// TIA Portal V16 export
// export: Created 2024-05-10T06:46:43.1229675Z, ExportSetting WithDefaults, DisplayName Totally Integrated Automation Portal, DisplayVersion V16, DisplayName TIA Portal Version Control Interface, DisplayVersion V16, DisplayName TIA Portal Openness, DisplayVersion V16, DisplayName STEP 7 Professional, DisplayVersion V16, DisplayName STEP 7 Safety, DisplayVersion V16, DisplayName WinCC Professional, DisplayVersion V16
FUNCTION_BLOCK "F121_SinaParaWrite(SV660F)"   // FB121, LAD
{ S7_Optimized_Access := 'TRUE' }
VERSION : 0.1
// stored: AutoNumber false, IsIECCheckEnabled false, IsRetainMemResEnabled false, MemoryReserve 100, SetENOAutomatically false, UDAEnableTagReadback false
   VAR_INPUT
      ID_回原高速 : DInt;
      ID_回原低速 : DInt;
      ID_点动速度 : DInt;
      ID_最高速度 : DInt;
      IM_故障复位 : Bool;
      ID_111报文标识符 { ExternalAccessible := 'False'; ExternalVisible := 'False'; ExternalWritable := 'False'} : HW_IO;
   END_VAR
   VAR_OUTPUT
      OM_准备好 : Bool;
      OM_进行中 : Bool;
      OM_正常完了 : Bool;
      OR_数据Real : Real;
      OD_数据Dint : DInt;
      OW_数据格式 : Int;
      OW_故障码 : Int;
      OM_故障 : Bool;
      OW_SFB调用错误 : Word;
   END_VAR
   VAR
      MT_Time { ExternalAccessible := 'False'; ExternalVisible := 'False'; ExternalWritable := 'False'} : IEC_TIMER;
   END_VAR
   VAR_TEMP
      MD_回原高速 : Array[1..2] of DInt;
      MD_回原低速 : Array[1..2] of DInt;
      MD_点动正速度 : Array[1..2] of DInt;
      MD_点动负速度 : Array[1..2] of DInt;
      MD_最高速度 : Array[1..2] of DInt;
      M_回原高速变更 : Bool;
      M_回原低速变更 : Bool;
      M_点动正速度变更 : Bool;
      M_点动负速度变更 : Bool;
      M_最高速度变更 : Bool;
      M_回原高速写入 : Bool;
      M_回原低速写入 : Bool;
      M_点动正速度写入 : Bool;
      M_点动负速度写入 : Bool;
      M_最高速度写入 : Bool;
      M_开始 : Bool;
      MW_Parameter : Int;
      MW_Index : Int;
      MD_Value : DInt;
      M_Pulse : Array[1..2] of Bool;
   END_VAR
   VAR_TEMP   // added for the SCL form of the ladder/FBD networks
      _w1 : Bool;
      _w2 : Bool;
      _w3 : Bool;
      _w4 : Bool;
      _w5 : Bool;
      _w6 : Bool;
   END_VAR
BEGIN

REGION Network 1: 回原高速
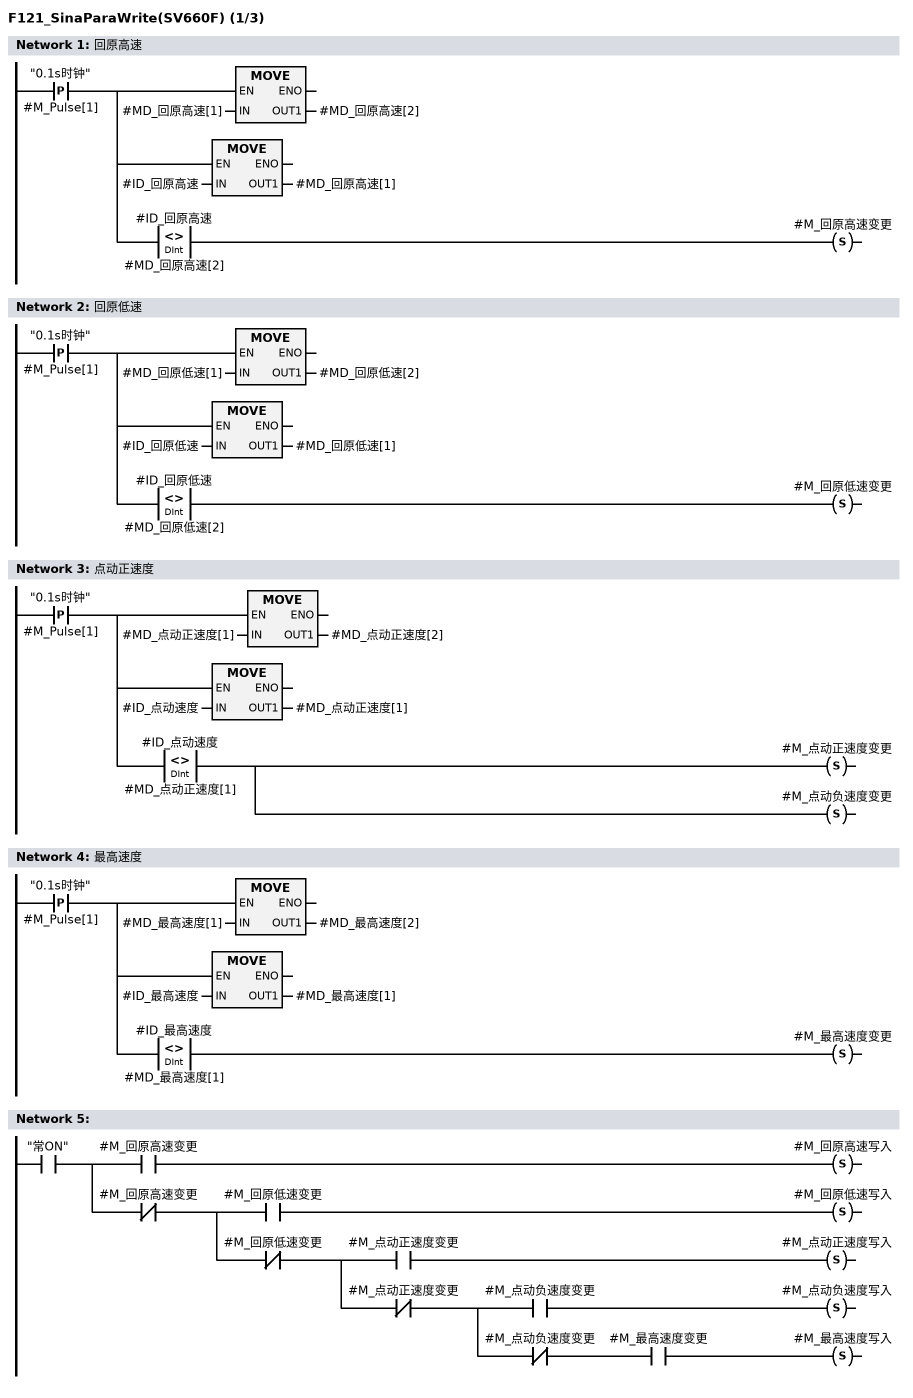
   RUNG wire#powerrail
      P_Contact(operand := "0.1s时钟", bit := #M_Pulse[1])
      wire#w1
      Move(in := #MD_回原高速[1], out1 => #MD_回原高速[2])
   END_RUNG
   RUNG wire#w1
      Move(in := #ID_回原高速, out1 => #MD_回原高速[1])
   END_RUNG
   RUNG wire#w1
      { S7_Templates := "SrcType := DInt" } NE_Contact(in1 := #ID_回原高速, in2 := #MD_回原高速[2])
      S_Coil( #M_回原高速变更 )
   END_RUNG
   // the same network as SCL:
   #_w1 := "0.1s时钟" AND NOT #M_Pulse[1];   // rising edge of "0.1s时钟"
   #M_Pulse[1] := "0.1s时钟";
   IF #_w1 THEN
       #MD_回原高速[2] := #MD_回原高速[1];
       #MD_回原高速[1] := #ID_回原高速;
   END_IF;
   IF #_w1 AND (#ID_回原高速 <> #MD_回原高速[2]) THEN #M_回原高速变更 := TRUE; END_IF;
END_REGION

REGION Network 2: 回原低速
   RUNG wire#powerrail
      P_Contact(operand := "0.1s时钟", bit := #M_Pulse[1])
      wire#w1
      Move(in := #MD_回原低速[1], out1 => #MD_回原低速[2])
   END_RUNG
   RUNG wire#w1
      Move(in := #ID_回原低速, out1 => #MD_回原低速[1])
   END_RUNG
   RUNG wire#w1
      { S7_Templates := "SrcType := DInt" } NE_Contact(in1 := #ID_回原低速, in2 := #MD_回原低速[2])
      S_Coil( #M_回原低速变更 )
   END_RUNG
   // the same network as SCL:
   #_w1 := "0.1s时钟" AND NOT #M_Pulse[1];   // rising edge of "0.1s时钟"
   #M_Pulse[1] := "0.1s时钟";
   IF #_w1 THEN
       #MD_回原低速[2] := #MD_回原低速[1];
       #MD_回原低速[1] := #ID_回原低速;
   END_IF;
   IF #_w1 AND (#ID_回原低速 <> #MD_回原低速[2]) THEN #M_回原低速变更 := TRUE; END_IF;
END_REGION

REGION Network 3: 点动正速度
   RUNG wire#powerrail
      P_Contact(operand := "0.1s时钟", bit := #M_Pulse[1])
      wire#w1
      Move(in := #MD_点动正速度[1], out1 => #MD_点动正速度[2])
   END_RUNG
   RUNG wire#w1
      Move(in := #ID_点动速度, out1 => #MD_点动正速度[1])
   END_RUNG
   RUNG wire#w1
      { S7_Templates := "SrcType := DInt" } NE_Contact(in1 := #ID_点动速度, in2 := #MD_点动正速度[1])
      wire#w2
      S_Coil( #M_点动正速度变更 )
   END_RUNG
   RUNG wire#w2
      S_Coil( #M_点动负速度变更 )
   END_RUNG
   // the same network as SCL:
   #_w1 := "0.1s时钟" AND NOT #M_Pulse[1];   // rising edge of "0.1s时钟"
   #M_Pulse[1] := "0.1s时钟";
   IF #_w1 THEN
       #MD_点动正速度[2] := #MD_点动正速度[1];
       #MD_点动正速度[1] := #ID_点动速度;
   END_IF;
   IF #_w1 AND (#ID_点动速度 <> #MD_点动正速度[1]) THEN
       #M_点动正速度变更 := TRUE;
       #M_点动负速度变更 := TRUE;
   END_IF;
END_REGION

REGION Network 4: 最高速度
   RUNG wire#powerrail
      P_Contact(operand := "0.1s时钟", bit := #M_Pulse[1])
      wire#w1
      Move(in := #MD_最高速度[1], out1 => #MD_最高速度[2])
   END_RUNG
   RUNG wire#w1
      Move(in := #ID_最高速度, out1 => #MD_最高速度[1])
   END_RUNG
   RUNG wire#w1
      { S7_Templates := "SrcType := DInt" } NE_Contact(in1 := #ID_最高速度, in2 := #MD_最高速度[1])
      S_Coil( #M_最高速度变更 )
   END_RUNG
   // the same network as SCL:
   #_w1 := "0.1s时钟" AND NOT #M_Pulse[1];   // rising edge of "0.1s时钟"
   #M_Pulse[1] := "0.1s时钟";
   IF #_w1 THEN
       #MD_最高速度[2] := #MD_最高速度[1];
       #MD_最高速度[1] := #ID_最高速度;
   END_IF;
   IF #_w1 AND (#ID_最高速度 <> #MD_最高速度[1]) THEN #M_最高速度变更 := TRUE; END_IF;
END_REGION

REGION Network 5
   RUNG wire#powerrail
      Contact( "常ON" )
      wire#w1
      Contact( #M_回原高速变更 )
      S_Coil( #M_回原高速写入 )
   END_RUNG
   RUNG wire#w1
      I_Contact( #M_回原高速变更 )
      wire#w2
      Contact( #M_回原低速变更 )
      S_Coil( #M_回原低速写入 )
   END_RUNG
   RUNG wire#w2
      I_Contact( #M_回原低速变更 )
      wire#w3
      Contact( #M_点动正速度变更 )
      S_Coil( #M_点动正速度写入 )
   END_RUNG
   RUNG wire#w3
      I_Contact( #M_点动正速度变更 )
      wire#w4
      Contact( #M_点动负速度变更 )
      S_Coil( #M_点动负速度写入 )
   END_RUNG
   RUNG wire#w4
      I_Contact( #M_点动负速度变更 )
      Contact( #M_最高速度变更 )
      S_Coil( #M_最高速度写入 )
   END_RUNG
   // the same network as SCL:
   IF "常ON" AND #M_回原高速变更 THEN #M_回原高速写入 := TRUE; END_IF;
   #_w1 := "常ON" AND NOT #M_回原高速变更;
   IF #_w1 AND #M_回原低速变更 THEN #M_回原低速写入 := TRUE; END_IF;
   #_w2 := #_w1 AND NOT #M_回原低速变更;
   IF #_w2 AND #M_点动正速度变更 THEN #M_点动正速度写入 := TRUE; END_IF;
   #_w3 := #_w2 AND NOT #M_点动正速度变更;
   IF #_w3 AND #M_点动负速度变更 THEN #M_点动负速度写入 := TRUE; END_IF;
   IF #_w3 AND NOT #M_点动负速度变更 AND #M_最高速度变更 THEN #M_最高速度写入 := TRUE; END_IF;
END_REGION

REGION Network 6
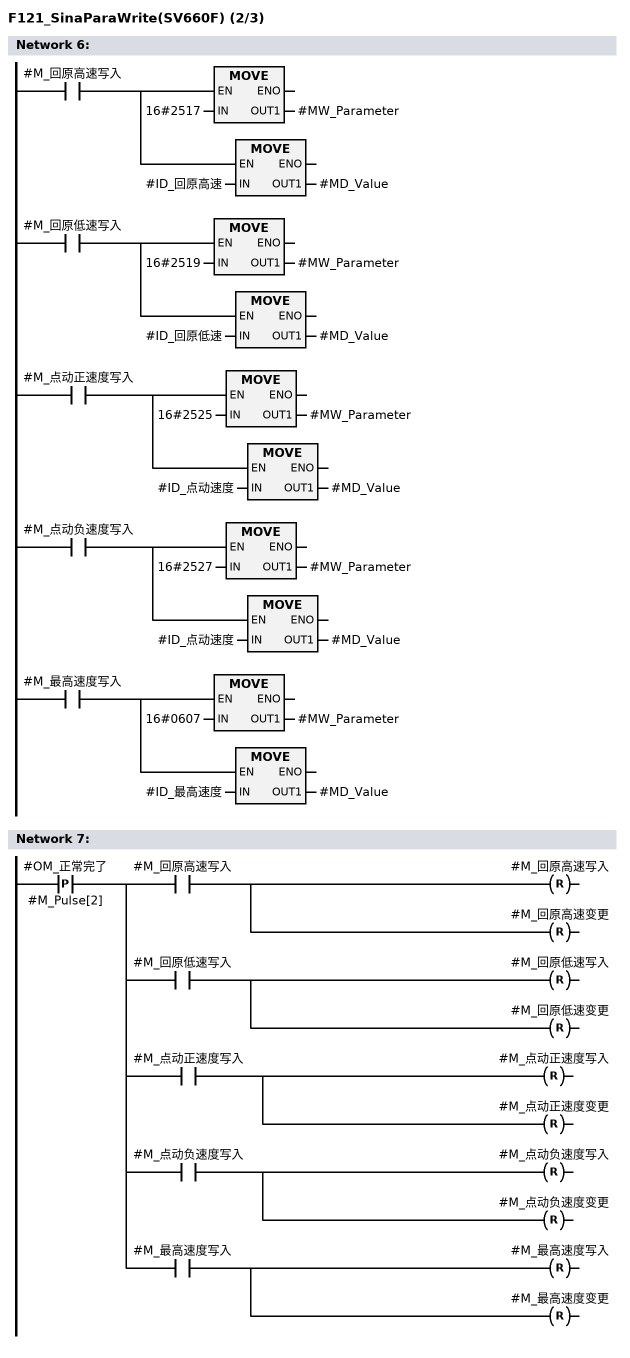
   RUNG wire#powerrail
      Contact( #M_回原高速写入 )
      wire#w1
      Move(in := 16#2517, out1 => #MW_Parameter)
   END_RUNG
   RUNG wire#w1
      Move(in := #ID_回原高速, out1 => #MD_Value)
   END_RUNG
   RUNG wire#powerrail
      Contact( #M_回原低速写入 )
      wire#w2
      Move(in := 16#2519, out1 => #MW_Parameter)
   END_RUNG
   RUNG wire#w2
      Move(in := #ID_回原低速, out1 => #MD_Value)
   END_RUNG
   RUNG wire#powerrail
      Contact( #M_点动正速度写入 )
      wire#w3
      Move(in := 16#2525, out1 => #MW_Parameter)
   END_RUNG
   RUNG wire#w3
      Move(in := #ID_点动速度, out1 => #MD_Value)
   END_RUNG
   RUNG wire#powerrail
      Contact( #M_点动负速度写入 )
      wire#w4
      Move(in := 16#2527, out1 => #MW_Parameter)
   END_RUNG
   RUNG wire#w4
      Move(in := #ID_点动速度, out1 => #MD_Value)
   END_RUNG
   RUNG wire#powerrail
      Contact( #M_最高速度写入 )
      wire#w5
      Move(in := 16#0607, out1 => #MW_Parameter)
   END_RUNG
   RUNG wire#w5
      Move(in := #ID_最高速度, out1 => #MD_Value)
   END_RUNG
   // the same network as SCL:
   IF #M_回原高速写入 THEN
       #MW_Parameter := 16#2517;
       #MD_Value := #ID_回原高速;
   END_IF;
   IF #M_回原低速写入 THEN
       #MW_Parameter := 16#2519;
       #MD_Value := #ID_回原低速;
   END_IF;
   IF #M_点动正速度写入 THEN
       #MW_Parameter := 16#2525;
       #MD_Value := #ID_点动速度;
   END_IF;
   IF #M_点动负速度写入 THEN
       #MW_Parameter := 16#2527;
       #MD_Value := #ID_点动速度;
   END_IF;
   IF #M_最高速度写入 THEN
       #MW_Parameter := 16#0607;
       #MD_Value := #ID_最高速度;
   END_IF;
END_REGION

REGION Network 7
   RUNG wire#powerrail
      P_Contact(operand := #OM_正常完了, bit := #M_Pulse[2])
      wire#w1
      Contact( #M_回原高速写入 )
      wire#w2
      R_Coil( #M_回原高速写入 )
   END_RUNG
   RUNG wire#w2
      R_Coil( #M_回原高速变更 )
   END_RUNG
   RUNG wire#w1
      Contact( #M_回原低速写入 )
      wire#w3
      R_Coil( #M_回原低速写入 )
   END_RUNG
   RUNG wire#w3
      R_Coil( #M_回原低速变更 )
   END_RUNG
   RUNG wire#w1
      Contact( #M_点动正速度写入 )
      wire#w4
      R_Coil( #M_点动正速度写入 )
   END_RUNG
   RUNG wire#w4
      R_Coil( #M_点动正速度变更 )
   END_RUNG
   RUNG wire#w1
      Contact( #M_点动负速度写入 )
      wire#w5
      R_Coil( #M_点动负速度写入 )
   END_RUNG
   RUNG wire#w5
      R_Coil( #M_点动负速度变更 )
   END_RUNG
   RUNG wire#w1
      Contact( #M_最高速度写入 )
      wire#w6
      R_Coil( #M_最高速度写入 )
   END_RUNG
   RUNG wire#w6
      R_Coil( #M_最高速度变更 )
   END_RUNG
   // the same network as SCL:
   #_w1 := #OM_正常完了 AND NOT #M_Pulse[2];   // rising edge of #OM_正常完了
   #M_Pulse[2] := #OM_正常完了;
   #_w2 := #_w1 AND #M_回原高速写入;
   IF #_w2 THEN
       #M_回原高速写入 := FALSE;
       #M_回原高速变更 := FALSE;
   END_IF;
   #_w3 := #_w1 AND #M_回原低速写入;
   IF #_w3 THEN
       #M_回原低速写入 := FALSE;
       #M_回原低速变更 := FALSE;
   END_IF;
   #_w4 := #_w1 AND #M_点动正速度写入;
   IF #_w4 THEN
       #M_点动正速度写入 := FALSE;
       #M_点动正速度变更 := FALSE;
   END_IF;
   #_w5 := #_w1 AND #M_点动负速度写入;
   IF #_w5 THEN
       #M_点动负速度写入 := FALSE;
       #M_点动负速度变更 := FALSE;
   END_IF;
   #_w6 := #_w1 AND #M_最高速度写入;
   IF #_w6 THEN
       #M_最高速度写入 := FALSE;
       #M_最高速度变更 := FALSE;
   END_IF;
END_REGION

REGION Network 8
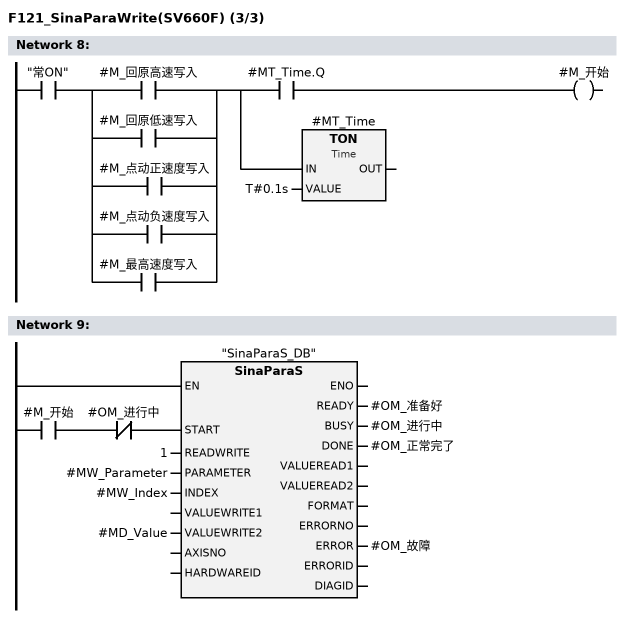
   #_w1 := "常ON" AND (#M_回原高速写入 OR #M_回原低速写入 OR #M_点动正速度写入 OR #M_点动负速度写入 OR #M_最高速度写入);
   #M_开始 := #_w1 AND #MT_Time.Q;
   #MT_Time.TON(IN := #_w1, PT := T#0.1s);   // TON coil
END_REGION

REGION Network 9
   RUNG wire#powerrail
      "SinaParaS_DB".SinaParaS(Start := wire#w1, ReadWrite := 1, Parameter := #MW_Parameter, Index := #MW_Index, ValueWrite1 :=, ValueWrite2 := #MD_Value, AxisNo :=, hardwareId :=, Ready => #OM_准备好, Busy => #OM_进行中, Done => #OM_正常完了, ValueRead1 =>, ValueRead2 =>, Format =>, ErrorNo =>, Error => #OM_故障, ErrorId =>, DiagId =>)
   END_RUNG
   RUNG wire#powerrail
      Contact( #M_开始 )
      I_Contact( #OM_进行中 )
   END_RUNG wire#w1
   // the same network as SCL:
   "SinaParaS_DB"(Start := #M_开始 AND NOT #OM_进行中,   // SinaParaS
                  ReadWrite := 1,
                  Parameter := #MW_Parameter,
                  Index := #MW_Index,
                  ValueWrite2 := #MD_Value,
                  Ready => #OM_准备好,
                  Busy => #OM_进行中,
                  Done => #OM_正常完了,
                  Error => #OM_故障);
END_REGION
END_FUNCTION_BLOCK
